// TIA Portal V17 export
// export: Created 2023-02-14T02:49:41.9158648Z, ExportSetting WithDefaults, DisplayName Totally Integrated Automation Portal, DisplayVersion V17, DisplayName TIA Portal Openness, DisplayVersion V17, DisplayName TIA Portal Teamcenter Gateway, DisplayVersion V17, DisplayName TIA Portal Version Control Interface, DisplayVersion V17, DisplayName SINAMICS Startdrive Advanced, DisplayVersion V17, DisplayName SINAMICS Startdrive G130, G150, S120, S150, SINAMICS MV, S210, DisplayVersion V17, DisplayName SINAMICS Startdrive G110M, G120, G120C, G120D, G120P, G115D, DisplayVersion V17, DisplayName STEP 7 Professional, DisplayVersion V17, DisplayName STEP 7 Safety, DisplayVersion V17, DisplayName WinCC Professional, DisplayVersion V17
DATA_BLOCK "T-51_HW"   // DB370
VERSION : 0.1
// stored: AutoNumber false, DBAccessibleFromOPCUA true, DBAccessibleFromWebserver true, InstanceOfName Hot_Water, InstanceOfType FB
"Hot_Water"
   // VAR_INPUT
   //    IN_FBAV_Inload : Bool;
   //    IN_FBAV_Outlet : Bool;
   //    IN_FBAV_Transfer : Bool;
   //    IN_FBP_Transfer : Bool;
   //    IN_FBP_Transfer_SP : Real;
   //    IN_Dose_Run : Bool;
   //    IN_Dose_Held : Bool;
   //    IN_Dose_Complete : Bool;
   //    IN_Dose_Header_1 : Bool;
   //    IN_Dose_Header_2 : Bool;
   //    IN_Dose_Valve_Cmd : Bool;
   //    IN_Dose_Pump_Cmd : Bool;
   //    IN_Dose_Pump_Sp : Real;
   //    IN_Dose_LineOK : Bool;
   //    IN_Low_Level : Bool;
   //    IN_Med_Level : Bool;
   //    IN_High_Level : Bool;
   //    IN_FBCV : Bool;
   //    "IN_FBCV_Act%" : Real;
   //    IN_Temperature : Real;
   // END_VAR
   // VAR_OUTPUT
   //    Out_AV_Inload : Bool;
   //    Out_AV_Outlet : Bool;
   //    Out_AV_Transfer : Bool;
   //    Out_P_Transfer : Bool;
   //    Out_P_Transfer_Sp : Real;
   //    OUT_CV : Bool;
   //    Out_Temp_Act : Real;
   //    Out_Temp_Sp : Real;
   // END_VAR
   // VAR
   //    Cmd : Struct
   //       Inload_Start : Bool;
   //       Inload_Mode : Bool;
   //       ReadyForTransfer : Bool;
   //       Transfer_Mode : Bool;
   //    END_STRUCT;
   // END_VAR
   // VAR RETAIN
   //    Param : Struct
   //       Temperature_SP : Real;
   //    END_STRUCT;
   // END_VAR
   // VAR
   //    State : Struct
   //       Tank_LL : Bool;
   //       Tank_ML : Bool;
   //       Tank_HL : Bool;
   //       Inload_EN : Bool;
   //       Inload_Aut : Bool;
   //       Inloading : Bool;
   //       Ready_For_Transfer_EN : Bool;
   //       Ready_For_Transfer : Bool;
   //       Tank_Available : Bool;
   //       Transfer_on_Prog : Bool;
   //    END_STRUCT;
   //    alwaysON : Bool;
   //    r : Struct
   //       PosE1 : Bool;
   //       PosE2 : Bool;
   //       PosE3 : Bool;
   //       PosE4 : Bool;
   //       PosE5 : Bool;
   //       PosE6 : Bool;
   //       PosE7 : Bool;
   //       PosE8 : Bool;
   //       PosE9 : Bool;
   //       PosE10 : Bool;
   //       PosE11 : Bool;
   //       PosE12 : Bool;
   //       PosE13 : Bool;
   //       PosE14 : Bool;
   //       PosE15 : Bool;
   //       PosE16 : Bool;
   //       PosE17 : Bool;
   //       PosE18 : Bool;
   //       PosE19 : Bool;
   //       PosE20 : Bool;
   //       PosE21 : Bool;
   //       PosE22 : Bool;
   //       PosE23 : Bool;
   //       PosE24 : Bool;
   //       PosE25 : Bool;
   //       PosE26 : Bool;
   //       PosE27 : Bool;
   //       PosE28 : Bool;
   //       PosE29 : Bool;
   //       PosE30 : Bool;
   //       PosE31 : Bool;
   //       PosE32 : Bool;
   //    END_STRUCT;
   //    Actuator : Struct
   //       AV_Inload : Bool;
   //       AV_Outlet : Bool;
   //       AV_Transfer : Bool;
   //       AV_CIP_Tank : Bool;
   //       AV_CIP_Line : Bool;
   //       P_Transfer : Bool;
   //       P_Inload : Bool;
   //       P_CIP : Bool;
   //       CV : Bool;
   //    END_STRUCT;
   //    SPumpTim { S7_SetPoint := 'True'} : TON_TIME;
   // END_VAR
BEGIN
END_DATA_BLOCK
